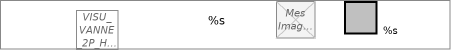
VISUALIZATION VISU_LIGNE_EAU  // 451x50
VAR_IN_OUT
	m_Input_LIGNE_EAU : BLOCK_LIGNE_REF;
END_VAR
    Polyline (451,20)
    Polyline (80,20)
    Polyline (129,20)
    Polygon (140,20)
    Polygon (317,20)
    Rectangle (380,15 65x31), "%s", text variable: m_Input_LIGNE_EAU.mnemo_DEX, invisible if: m_Input_LIGNE_EAU.CONF_NO_DexT
    Group (344,1 33x33), invisible if: (m_Input_LIGNE_EAU.CONF_NO_DexT) <> 0
        Rectangle (0,0 33x33), colour toggle: (m_Input_LIGNE_EAU.IN_DExT) <> 0
        Polyline (16,8)
        Polyline (24,15)
    Rectangle (154,5 125x31), "%s", text variable: m_Input_LIGNE_EAU.mnemo
    Frame (76,10 42x40)
        shows VISU_VANNE_2P_H_ACT2(m_Input_VANNE := m_Input_LIGNE_EAU.VEx)
        p1022016623: m_Input_LIGNE_EAU.VEx
    Image (276,1 39x37), invisible if: NOT m_Input_LIGNE_EAU.STATE_NOK, image: MesImages.warning
END_VISUALIZATION

(* stored: Version 1.1.0.1, ProductVersion 3.1.4024.10
   Visu VISU_LIGNE_EAU: Id {b8009b82-a36f-467b-843b-affc2c692e74} *)
